FUNCTION_BLOCK FB_Machine
VAR
	fbArm				: FB_Arm;
	
	(*Button*)
	btStartHoming		: BOOL;
	rHighSpeedHzValue	: REAL;
	rLowSpeedHzValue	: REAL;
	rHzToRawRatioValue	: REAL;
	tDelayTimeValue		: TIME;
END_VAR

fbArm.Homing(btStartHoming);
fbArm.HighSpeedHz := rHighSpeedHzValue;
fbArm.LowSpeedHz := rLowSpeedHzValue;
fbArm.HzToRawRatio := rHzToRawRatioValue;
fbArm.DelayTime := tDelayTimeValue;

END_FUNCTION_BLOCK

(* stored: Version 1.1.0.1, ProductVersion 3.1.4024.12
   POU FB_Machine: Id {0762e580-feee-46d7-a51d-4d74e4f1fd72}, SpecialFunc None *)
